INTERFACE Callable

METHOD call : Awaitable
VAR_INPUT
	callback: Callback;
END_VAR
END_METHOD

END_INTERFACE

(* stored: Version 1.1.0.1, ProductVersion 3.1.4024.12
   Itf Callable: Id {e88c15c0-c2f3-4df0-aeff-6b1db87e104a}
   Method call: Id {2fff1301-c33b-416e-8617-f1edcda4748a} *)
